{attribute 'GeneratedUsingTerminal: EK1100-0000-0018'}
{attribute addProperty BoxType "EK1100-0000-0018"}
{attribute addProperty Id "StateAT %I*UINT2"}
{attribute addProperty CRC "1863965483"}
{attribute addProperty Size "2"}
TYPE InfoData_6F19DB2B :
STRUCT
	{attribute addProperty Name "State"}
	State AT %I* : UINT;
END_STRUCT
END_TYPE

(* stored: Version 1.2.0.0, ProductVersion 3.1.4024.9
   DUT InfoData_6F19DB2B: Id {78e3193b-c632-40ed-8236-3de50d015845} *)
